{attribute addProperty BoxType "EL7342-0000-0023"}
{attribute addProperty Id "EnableBIT10.1251ResetBIT10.1252Reduce_torqueBIT10.1253Threshold_activeBIT10.1254"}
{attribute addProperty CRC "3530893112"}
{attribute addProperty SizeInBites "16"}
{attribute addProperty SizeInBytes "2"}
TYPE Control_D2752738 :
STRUCT
	{attribute addProperty Name "Enable"}
	Enable : BIT;
	{attribute addProperty Name "Reset"}
	Reset : BIT;
	{attribute addProperty Name "Reduce_torque"}
	Reduce_torque : BIT;
	{attribute addProperty Name "Threshold_active"}
	Threshold_active : BIT;
	{attribute 'hide'}
	reserve_1_BIT_0 : BIT;
	{attribute 'hide'}
	reserve_1_BIT_1 : BIT;
	{attribute 'hide'}
	reserve_1_BIT_2 : BIT;
	{attribute 'hide'}
	reserve_1_BIT_3 : BIT;
	{attribute 'hide'}
	reserve_2 : BYTE;
END_STRUCT
END_TYPE

(* stored: Version 1.2.0.0, ProductVersion 3.1.4024.9
   DUT Control_D2752738: Id {1efcf8db-dc2b-496a-b746-d7e30f63194a} *)
